// TIA Portal V16 export
DATA_BLOCK "DB_Conveyor_LAD"   // DB2
{ S7_Optimized_Access := 'TRUE' }
// stored: AutoNumber false, InstanceOfName FB_Conveyor_LAD, InstanceOfNumber 2, InstanceOfType FB, ReadOnly false
"FB_Conveyor_LAD"
BEGIN
END_DATA_BLOCK
